// TIA Portal V17 export
// export: Created 2023-12-22T15:08:02.7286606Z, ExportSetting WithDefaults, DisplayName Totally Integrated Automation Portal, DisplayVersion V17, DisplayName TIA Portal Openness, DisplayVersion V17, DisplayName TIA Portal Version Control Interface, DisplayVersion V17, DisplayName STEP 7 Professional, DisplayVersion V17, DisplayName STEP 7 Safety, DisplayVersion V17, DisplayName WinCC Advanced, DisplayVersion V17
FUNCTION_BLOCK "PIDx"   // FB260, LAD
{ S7_Optimized_Access := 'TRUE' }
VERSION : 0.1
// stored: AutoNumber false, IsIECCheckEnabled false, IsRetainMemResEnabled false, MemoryReserve 100, SetENOAutomatically false, UDAEnableTagReadback false
   VAR DB_SPECIFIC
      Time_DTL { S7_SetPoint := 'True'} : DTL;
   END_VAR
   VAR_TEMP   // added for the SCL form of the ladder/FBD networks
      _w1 : Bool;
      _w2 : Bool;
   END_VAR
BEGIN

REGION Network 1: Основной регулятор по давлению
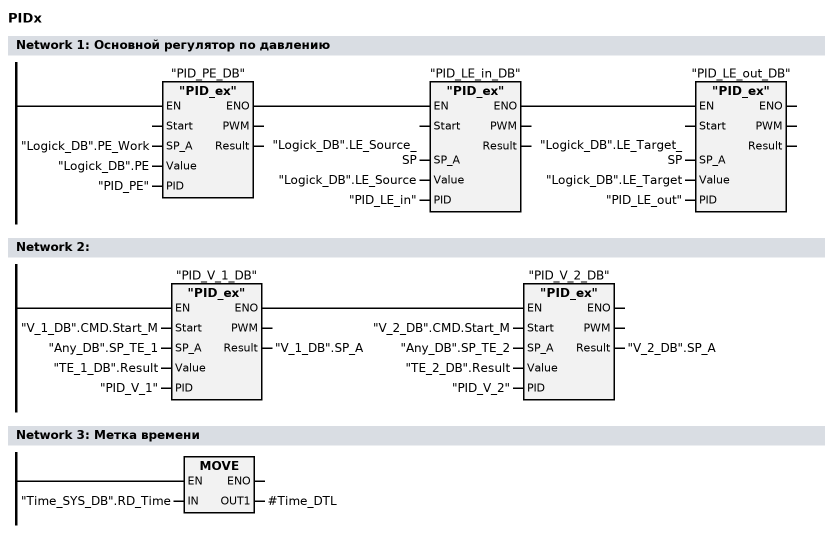
   RUNG wire#powerrail
      "PID_PE_DB"(Start :=, SP_A := "Logick_DB".PE_Work, Value := "Logick_DB".PE, PID := "PID_PE", PWM =>, Result =>)
      "PID_LE_in_DB"(Start :=, SP_A := "Logick_DB".LE_Source_SP, Value := "Logick_DB".LE_Source, PID := "PID_LE_in", PWM =>, Result =>)
      "PID_LE_out_DB"(Start :=, SP_A := "Logick_DB".LE_Target_SP, Value := "Logick_DB".LE_Target, PID := "PID_LE_out", PWM =>, Result =>)
   END_RUNG
   // the same network as SCL:
   "PID_PE_DB"(SP_A := "Logick_DB".PE_Work, Value := "Logick_DB".PE, PID := "PID_PE", ENO => #_w1);   // "PID_ex"
   "PID_LE_in_DB"(EN := #_w1,   // "PID_ex"
                  SP_A := "Logick_DB".LE_Source_SP,
                  Value := "Logick_DB".LE_Source,
                  PID := "PID_LE_in",
                  ENO => #_w2);
   IF #_w2 THEN
       "PID_LE_out_DB"(SP_A := "Logick_DB".LE_Target_SP, Value := "Logick_DB".LE_Target, PID := "PID_LE_out");   // "PID_ex"
   END_IF;
END_REGION

REGION Network 2
   RUNG wire#powerrail
      "PID_V_1_DB"(Start := "V_1_DB".CMD.Start_M, SP_A := "Any_DB".SP_TE_1, Value := "TE_1_DB".Result, PID := "PID_V_1", PWM =>, Result => "V_1_DB".SP_A)
      "PID_V_2_DB"(Start := "V_2_DB".CMD.Start_M, SP_A := "Any_DB".SP_TE_2, Value := "TE_2_DB".Result, PID := "PID_V_2", PWM =>, Result => "V_2_DB".SP_A)
   END_RUNG
   // the same network as SCL:
   "PID_V_1_DB"(Start := "V_1_DB".CMD.Start_M,   // "PID_ex"
                SP_A := "Any_DB".SP_TE_1,
                Value := "TE_1_DB".Result,
                PID := "PID_V_1",
                Result => "V_1_DB".SP_A,
                ENO => #_w1);
   IF #_w1 THEN
       "PID_V_2_DB"(Start := "V_2_DB".CMD.Start_M,   // "PID_ex"
                    SP_A := "Any_DB".SP_TE_2,
                    Value := "TE_2_DB".Result,
                    PID := "PID_V_2",
                    Result => "V_2_DB".SP_A);
   END_IF;
END_REGION

REGION Network 3: Метка времени
   RUNG wire#powerrail
      Move(in := "Time_SYS_DB".RD_Time, out1 => #Time_DTL)
   END_RUNG
   // the same network as SCL:
   #Time_DTL := "Time_SYS_DB".RD_Time;
END_REGION
END_FUNCTION_BLOCK
